// Mitsubishi GX Works2 project: selo com desliga   PLC: Q03UDV

PROGRAM MAIN
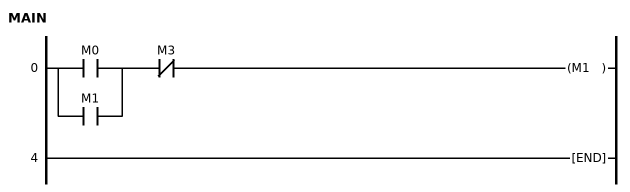
0     LD      M0
      OR      M1
      ANI     M3
      OUT     M1
4     END
END_PROGRAM
